{attribute 'hide_all_locals' := ''}
PROGRAM RET_COMMON
VAR_INPUT
	/// Zykluszeit Main-Task
	fDt: REAL := 0.001;
END_VAR

END_PROGRAM

(* stored: Version 1.1.0.1, ProductVersion 3.1.4024.12
   POU RET_COMMON: Id {371f0054-3649-4ee2-83d9-b6a67901040c}, SpecialFunc None *)
